INTERFACE IEnumerator EXTENDS IObject

// Shows curent collection element
PROPERTY ABSTRACT Current : PVOID
GET
END_GET
END_PROPERTY

// Moves Current pointer to next collection element
METHOD MoveNext : BOOL
END_METHOD

// Sets the enumerator to its initial position, which is before the first element in the collection
METHOD Reset
END_METHOD

END_INTERFACE

(* stored: Version 1.1.0.1
   Itf IEnumerator: Id {003d33a5-070b-07a7-317a-b66cff06678f}
   Property Current: Id {0e28ad9d-3061-0fd1-1451-fffc6356654b}
   Get Get: Id {f385e541-58c2-036e-3083-5b9dd71f64a7}
   Method MoveNext: Id {548c4f21-9b3a-0f8a-34fc-95200e15899c}
   Method Reset: Id {ed65fb3d-55e2-06ca-1906-cc193c654313} *)
